FUNCTION_BLOCK E_SPLIT (* Split an event *)
  (* Standard: 61499-2 *)
  (* Version 0.1, 2006-04-25, JHC, Holobloc Inc, Corrected ECC layout. *)
  (* Version 0.0, 2000-10-17, JHC, Rockwell Automation *)
  (* Compiler header: package fb.rt.events; *)
  (* Compiler Java Sun JDK 1.5.0 *)
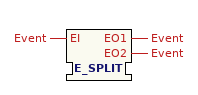
  EVENT_INPUT
    EI; (* Input event *)
  END_EVENT
  EVENT_OUTPUT
    EO1; (* First output event *)
    EO2; (* Second output event,etc. *)
  END_EVENT
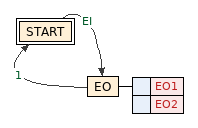
  EC_STATES
    START; (* Initial State *)
    EO : -> EO1, -> EO2; (* Output first,second event,etc. *)
  END_STATES
  EC_TRANSITIONS
    START TO EO := EI;
    EO TO START := 1;
  END_TRANSITIONS
END_FUNCTION_BLOCK
